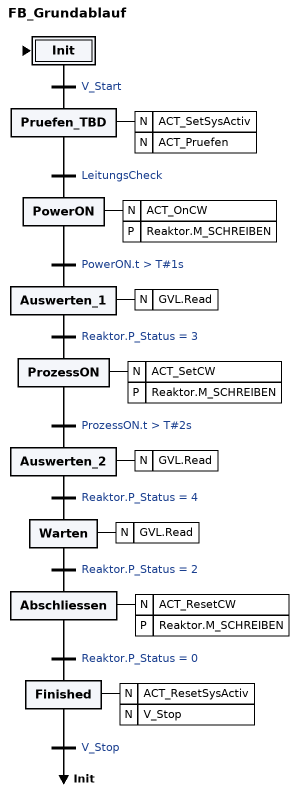
INITIAL_STEP Init:
END_STEP
TRANSITION FROM Init TO Pruefen_TBD
    := V_Start;
END_TRANSITION
STEP Pruefen_TBD:
    ACT_SetSysActiv(N);
    ACT_Pruefen(N);
END_STEP
TRANSITION FROM Pruefen_TBD TO PowerON
    := LeitungsCheck;
END_TRANSITION
STEP PowerON:
    ACT_OnCW(N);
    Reaktor.M_SCHREIBEN(P);
END_STEP
TRANSITION FROM PowerON TO Auswerten_1
    := PowerON.t > T#1s;
END_TRANSITION
STEP Auswerten_1:
    GVL.Read(N);
END_STEP
TRANSITION FROM Auswerten_1 TO ProzessON
    := Reaktor.P_Status = 3;
END_TRANSITION
STEP ProzessON:
    ACT_SetCW(N);
    Reaktor.M_SCHREIBEN(P);
END_STEP
TRANSITION FROM ProzessON TO Auswerten_2
    := ProzessON.t > T#2s;
END_TRANSITION
STEP Auswerten_2:
    GVL.Read(N);
END_STEP
TRANSITION FROM Auswerten_2 TO Warten
    := Reaktor.P_Status = 4;
END_TRANSITION
STEP Warten:
    GVL.Read(N);
END_STEP
TRANSITION FROM Warten TO Abschliessen
    := Reaktor.P_Status = 2;
END_TRANSITION
STEP Abschliessen:
    ACT_ResetCW(N);
    Reaktor.M_SCHREIBEN(P);
END_STEP
TRANSITION FROM Abschliessen TO Finished
    := Reaktor.P_Status = 0;
END_TRANSITION
STEP Finished:
    ACT_ResetSysActiv(N);
    V_Stop(N);
END_STEP
TRANSITION FROM Finished TO Init
    := V_Stop;
END_TRANSITION

ACTION ACT_OnCW:
CW.PowerOn := TRUE;
END_ACTION

ACTION ACT_Pruefen:
// TBD
END_ACTION

ACTION ACT_ResetCW:
CW.PowerOn := FALSE;
CW.SekReakt := 0;
CW.Leitung := 0;
CW.Temp := 0;
CW.Enlteermenge := 0;
CW.Pumpmenge := 0;
CW.Haltedauer := 0;
CW.Ruehrdauer := 0;
CW.Wartedauer := 0;
CW.Zirkulierdauer := 0;
END_ACTION

ACTION ACT_ResetSysActiv:
GVL.SysState := 1;
END_ACTION

ACTION ACT_SetCW:
CW.SekReakt := SekReakt;
CW.Leitung := Leitung;
CW.Temp := Temp;
CW.Enlteermenge := Entleermenge;
CW.Pumpmenge := Pumpmenge;
CW.Haltedauer := Haltedauer;
CW.Ruehrdauer := Ruehrdauer;
CW.Wartedauer := Wartedauer;
CW.Zirkulierdauer := Zirkulierdauer;
END_ACTION

ACTION ACT_SetSysActiv:
GVL.SysState := 2;
END_ACTION

END_FUNCTION_BLOCK

// ---- GlobalTextList.TcGTLO
TEXTLIST GlobalTextList
  594 = '"KeepAlive" der Kommunikation'
  213 = '%04x'
  656 = '%i'
  82 = '%s'
  105 = 'Act'
  5 = 'Activate'
  520 = 'Auffüllprozess läuft'
  842 = 'Auschalten'
  551 = 'Ausführen von Kommunikation'
  820 = 'Ausführen von Kommunikationsbefehl'
  888 = 'Ausschalten'
  177 = 'Busy:'
  154 = 'Client resetten'
  41 = 'Client zurücksetzen'
  364 = 'Connect'
  431 = 'Connected:'
  123 = 'ConnectionState'
  369 = 'ConnentionStatus'
  716 = 'ConnentionStatus:'
  988 = 'Controll-Word'
  676 = 'Controll-Word-Reaktor 1'
  461 = 'Debug-HMI'
  776 = 'Definiert welche Leitung verwendet wird'
  578 = 'Definierte Temperatur für Heiz- / Kühlprozess'
  47 = 'Definierter sekundär-Reaktor'
  35 = 'Disconnect'
  587 = 'Eigenschaften & Inputs'
  856 = 'Einschalten'
  668 = 'Enleermenge'
  20 = 'Entleerprozess läuft'
  519 = 'Error:'
  751 = 'Errorhandling'
  292 = 'ErrorID:'
  426 = 'Feldgerät-Steuerung'
  496 = 'Füllstandsensor'
  372 = 'GF1Activ'
  913 = 'GF2Activ'
  524 = 'GF3Activ'
  479 = 'GF4Activ'
  606 = 'GF5Activ'
  300 = 'GF6Activ'
  505 = 'GF7Activ'
  571 = 'GF8Activ'
  534 = 'Haltedauer'
  600 = 'Halteprozess läuft'
  705 = 'Heiz- / Kühlprozess läuft'
  42 = 'HK-System'
  828 = 'Input-Signal:'
  942 = 'Leitung'
  581 = 'Lesen'
  1134 = 'Messwert:'
  242 = 'Modus'
  924 = 'NameSpaceIndex:'
  907 = 'NodeID'
  136 = 'OPC UA'
  932 = 'POWER:'
  450 = 'PrimeActiv'
  282 = 'PrimReady'
  351 = 'Primärreaktor führt Prozess aus'
  770 = 'Primärreaktor ist bereit für den Prozess'
  331 = 'Pumpe'
  722 = 'Pumpmenge'
  152 = 'Pumpprozess läuft'
  1029 = 'P_DefTemp:'
  323 = 'P_MaxDrz:'
  1036 = 'ReactActiv'
  835 = 'ReactReady'
  297 = 'Reaktor 1'
  76 = 'Reaktor 2'
  509 = 'Reaktor 3'
  653 = 'Reaktor 4'
  173 = 'Reaktor 5'
  70 = 'Reaktor 6'
  444 = 'Reaktor 7'
  914 = 'Reaktor_1'
  946 = 'Ruehrdauer'
  933 = 'Rührer'
  40 = 'Rührprozess läuft'
  638 = 'Schreiben von Variablen zulassen'
  616 = 'SekActiv'
  650 = 'SekReady'
  373 = 'SekReakt'
  560 = 'Sekundärreaktor führt Prozess aus'
  923 = 'Sekundärreaktor ist bereit für den Prozess'
  701 = 'ServerState:'
  860 = 'Start'
  857 = 'Start sekundär Reaktor'
  291 = 'Start: Rezept'
  979 = 'Status-Word'
  421 = 'Status-Word-R1'
  183 = 'Status-Word-R2'
  447 = 'SysActiv'
  535 = 'SysReady'
  973 = 'Temp'
  27 = 'Temperatursensor'
  976 = 'Test-HMI'
  234 = 'Variablen werden gelese / beschrieben'
  320 = 'Verbinden mit Client'
  643 = 'Verbindung zum Server wurde erstellt'
  834 = 'VERBUNDEN:'
  972 = 'Verbunden: '
  889 = 'Wartedauer'
  362 = 'Warteprozess läuft'
  438 = 'Wie lange soll gerührt werden'
  301 = 'Wie lange soll gerührt werden '
  394 = 'Wie lange soll Temperatur gehalten werden'
  666 = 'Wie lange soll zirkuliert werden'
  768 = 'Zierkulierdauer'
  926 = 'Zirkulierprozess läuft'
  26 = 'Zu entleerende Menge'
  164 = 'Zu pumpende Menge'
  448 = 'Zustand'
END_TEXTLIST

// ---- VISUs/Test_Visu.TcVIS
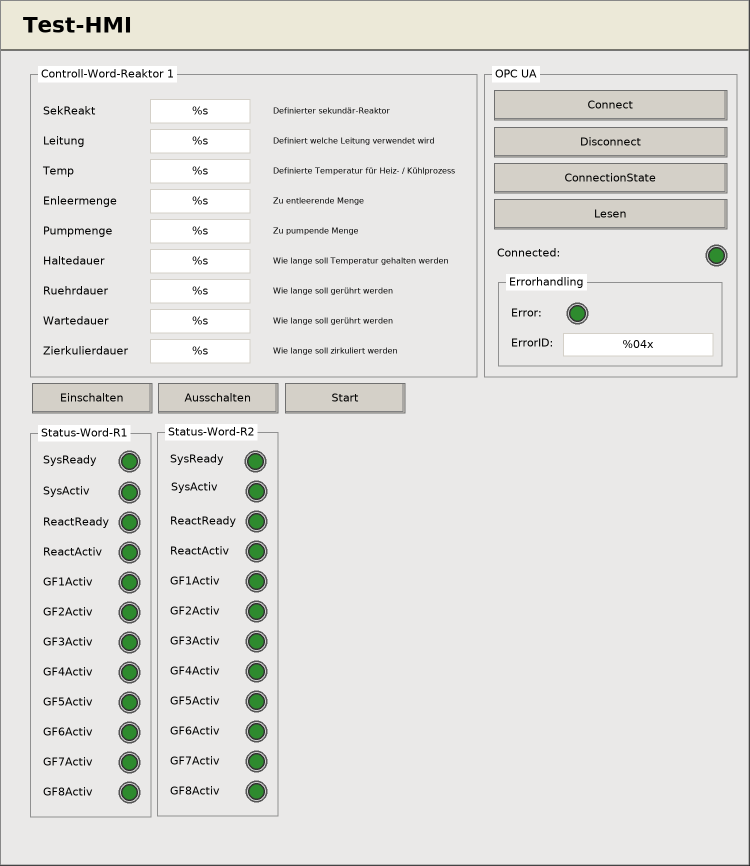
VISUALIZATION Test_Visu  // 750x866
    Rectangle (0,6 750x860)
    Rectangle (0,0 750x50)
    Label (20,0 480x50), "Test-HMI"
    GroupBox (30,66 447x311), "Controll-Word-Reaktor 1"
        Label (10,30 150x30), "SekReakt"
        Label (10,60 150x30), "Leitung"
        Label (10,90 150x30), "Temp"
        Label (10,120 150x30), "Enleermenge"
        Label (10,150 150x30), "Pumpmenge"
        Label (10,180 150x30), "Haltedauer"
        Label (10,210 150x30), "Ruehrdauer"
        Label (10,240 150x30), "Wartedauer"
        Label (10,270 150x30), "Zierkulierdauer"
        Textfield (120,33 100x24), "%s", text variable: GVL.R1_CW.SekReakt
            OnMouseClick: write GVL.R1_CW.SekReakt via Edit
        Textfield (120,63 100x24), "%s", text variable: GVL.R1_CW.Leitung
            OnMouseClick: write GVL.R1_CW.Leitung via Edit
        Textfield (120,93 100x24), "%s", text variable: GVL.R1_CW.Temp
            OnMouseClick: write GVL.R1_CW.Temp via Default
        Textfield (120,123 100x24), "%s", text variable: GVL.R1_CW.Enlteermenge
            OnMouseClick: write GVL.R1_CW.Enlteermenge via Edit
        Textfield (120,153 100x24), "%s", text variable: GVL.R1_CW.Pumpmenge
            OnMouseClick: write GVL.R1_CW.Pumpmenge via Edit
        Textfield (120,183 100x24), "%s", text variable: GVL.R1_CW.Haltedauer
            OnMouseClick: write GVL.R1_CW.Haltedauer via Edit
        Textfield (120,213 100x24), "%s", text variable: GVL.R1_CW.Ruehrdauer
            OnMouseClick: write GVL.R1_CW.Ruehrdauer via Edit
        Textfield (120,243 100x24), "%s", text variable: GVL.R1_CW.Wartedauer
            OnMouseClick: write GVL.R1_CW.Wartedauer via Edit
        Textfield (120,273 100x24), "%s", text variable: GVL.R1_CW.Zirkulierdauer
            OnMouseClick: write GVL.R1_CW.Zirkulierdauer via Edit
        Label (240,30 300x30), "Definierter sekundär-Reaktor"
        Label (240,60 300x30), "Definiert welche Leitung verwendet wird"
        Label (240,90 300x30), "Definierte Temperatur für Heiz- / Kühlprozess"
        Label (240,120 300x30), "Zu entleerende Menge"
        Label (240,150 300x30), "Zu pumpende Menge"
        Label (240,180 300x30), "Wie lange soll Temperatur gehalten werden"
        Label (240,210 300x30), "Wie lange soll gerührt werden"
        Label (240,240 300x30), "Wie lange soll gerührt werden"
        Label (240,270 300x30), "Wie lange soll zirkuliert werden"
    GroupBox (30,425 121x392), "Status-Word-R1"
        Label (10,82 150x30), "ReactReady"
        Label (10,112 150x30), "ReactActiv"
        Label (10,142 150x30), "GF1Activ"
        Label (10,172 150x30), "GF2Activ"
        Label (10,202 150x30), "GF3Activ"
        Label (10,232 150x30), "GF4Activ"
        Label (10,262 150x30), "GF5Activ"
        Label (10,292 150x30), "GF6Activ"
        Label (10,322 150x30), "GF7Activ"
        Label (10,352 150x30), "GF8Activ"
        Lamp1 (87,85 25x25), variable: GVL.R1_SW.ReactReady, style: Lamp-Lamp1-Green
        Lamp1 (87,115 25x25), variable: GVL.R1_SW.ReactActiv, style: Lamp-Lamp1-Green
        Lamp1 (87,145 25x25), variable: GVL.R1_SW.GF1Activ, style: Lamp-Lamp1-Green
        Lamp1 (87,175 25x25), variable: GVL.R1_SW.GF2Activ, style: Lamp-Lamp1-Green
        Lamp1 (87,205 25x25), variable: GVL.R1_SW.GF3Activ, style: Lamp-Lamp1-Green
        Lamp1 (87,235 25x25), variable: GVL.R1_SW.GF4Activ, style: Lamp-Lamp1-Green
        Lamp1 (87,265 25x25), variable: GVL.R1_SW.GF5Activ, style: Lamp-Lamp1-Green
        Lamp1 (87,295 25x25), variable: GVL.R1_SW.GF6Activ, style: Lamp-Lamp1-Green
        Lamp1 (87,325 25x25), variable: GVL.R1_SW.GF7Activ, style: Lamp-Lamp1-Green
        Lamp1 (87,355 25x25), variable: GVL.R1_SW.GF8Activ, style: Lamp-Lamp1-Green
        Lamp1 (87,55 25x25), variable: GVL.R1_SW.SysActiv, style: Lamp-Lamp1-Green
        Label (10,20 58x30), "SysReady"
    Button (32,383 120x30), "Einschalten"
        OnMouseClick: execute { GVL.R1_CW.PowerOn := 1; Reaktoranlage.R1.M_SCHREIBEN(); }
    GroupBox (484,66 253x311), "OPC UA"
        Button (10,24 233x30), "Connect"
            tap GVL.Connect
        GroupBox (14,208 224x92), "Errorhandling"
            Label (10,24 150x30), "Error:"
            Label (10,54 150x30), "ErrorID:"
            Lamp1 (67,27 25x25), variable: GVL.Error, style: Lamp-Lamp1-Green
            Textfield (65,59 150x23), "%04x", text variable: GVL.ErrorID, input disabled if: TRUE
        Button (10,61 233x30), "Disconnect"
            tap GVL.Disconnect
        Button (10,97 233x30), "ConnectionState"
            OnMouseClick: execute { Reaktoranlage.R1.M_ZUSTAND(); }
        Label (10,172 150x30), "Connected:"
        Lamp1 (220,177 25x25), variable: Reaktoranlage.R1.O_Verbunden, style: Lamp-Lamp1-Green
        Button (10,133 233x30), "Lesen"
            OnMouseClick: execute { Reaktoranlage.R1.M_Lesen(); }
    Label (40,476 58x30), "SysActiv"
    Button (158,383 120x30), "Ausschalten"
        OnMouseClick: execute { GVL.R1_CW.PowerOn := 0; Reaktoranlage.R1.M_SCHREIBEN(); }
    Button (285,383 120x30), "Start"
        tap GVL.Start
    Lamp1 (117,449 25x25), variable: GVL.R1_SW.SysReady, style: Lamp-Lamp1-Green
    GroupBox (157,424 121x392), "Status-Word-R2"
        Label (10,82 150x30), "ReactReady"
        Label (10,112 150x30), "ReactActiv"
        Label (10,142 150x30), "GF1Activ"
        Label (10,172 150x30), "GF2Activ"
        Label (10,202 150x30), "GF3Activ"
        Label (10,232 150x30), "GF4Activ"
        Label (10,262 150x30), "GF5Activ"
        Label (10,292 150x30), "GF6Activ"
        Label (10,322 150x30), "GF7Activ"
        Label (10,352 150x30), "GF8Activ"
        Lamp1 (87,85 25x25), variable: GVL.R2_SW.ReactReady, style: Lamp-Lamp1-Green
        Lamp1 (87,115 25x25), variable: GVL.R2_SW.ReactActiv, style: Lamp-Lamp1-Green
        Lamp1 (87,145 25x25), variable: GVL.R2_SW.GF1Activ, style: Lamp-Lamp1-Green
        Lamp1 (87,175 25x25), variable: GVL.R2_SW.GF2Activ, style: Lamp-Lamp1-Green
        Lamp1 (87,205 25x25), variable: GVL.R2_SW.GF3Activ, style: Lamp-Lamp1-Green
        Lamp1 (87,235 25x25), variable: GVL.R2_SW.GF4Activ, style: Lamp-Lamp1-Green
        Lamp1 (87,265 25x25), variable: GVL.R2_SW.GF5Activ, style: Lamp-Lamp1-Green
        Lamp1 (87,295 25x25), variable: GVL.R2_SW.GF6Activ, style: Lamp-Lamp1-Green
        Lamp1 (87,325 25x25), variable: GVL.R2_SW.GF7Activ, style: Lamp-Lamp1-Green
        Lamp1 (87,355 25x25), variable: GVL.R2_SW.GF8Activ, style: Lamp-Lamp1-Green
        Lamp1 (87,55 25x25), variable: GVL.R2_SW.SysActiv, style: Lamp-Lamp1-Green
        Label (10,20 58x30), "SysReady"
        Label (11,48 58x30), "SysActiv"
    Lamp1 (243,449 25x25), variable: GVL.R2_SW.SysActiv, style: Lamp-Lamp1-Green
END_VISUALIZATION
